FUNCTION_BLOCK DISTRIBUTION (* Basic FB with empty ECC *)
  (* Standard: 61499-2 *)
  (* Version 1.0, 2020-10-21, chong *)
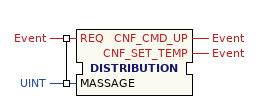
  EVENT_INPUT
    REQ WITH MASSAGE;
  END_EVENT
  EVENT_OUTPUT
    CNF_CMD_UP;
    CNF_SET_TEMP;
  END_EVENT
  VAR_INPUT
    MASSAGE : UINT;
  END_VAR
  EC_STATES
    START; (* Initial State *)
  END_STATES
END_FUNCTION_BLOCK
